PROGRAM MAIN
VAR
END_VAR

RunGrindingWheel ();

END_PROGRAM

(* stored: Version 1.1.0.1, ProductVersion 3.1.4024.4
   POU MAIN: Id {f64c6a75-415f-4ac2-91f2-2395a924fc72}, SpecialFunc None *)
